(* IEC 61131-3 sources: SerComm/, 4 files *)

(* ---- SerComm.typ ---- *)
(********************************************************************
 * COPYRIGHT -- Automation Resources Group
 ********************************************************************
 * Library: SerComm
 * File: SerComm.typ
 * Author: David Blackburn
 * Created: June 21, 2013
 ********************************************************************
 * Data types of library SerComm
 ********************************************************************)

TYPE

END_TYPE

(* ---- SerialCommMgr.typ ---- *)
(*
 * File: SerialCommMgr.typ
 * Copyright (c) 2023 Loupe
 * https://loupe.team
 *
 * This file is part of SerComm, licensed under the MIT License.
 *
 *)

TYPE
	SERCOMM_ERR_enum :
		(
		SERCOMM_ERR_INVALIDINPUT := 50000,
		SERCOMM_ERR_RECVDATATOOLARGE,
		SERCOMM_ERR_SENDDATATOOLARGE,
		SERCOMM_ERR_
		);
	SERCOMM_ST_enum :
		(
		SERCOMM_ST_CLOSED,
		SERCOMM_ST_OPENING,
		SERCOMM_ST_RUNNING,
		SERCOMM_ST_CLOSING,
		SERCOMM_ST_ERROR
		);
	SERCOMM_RECV_ST_enum :
		(
		SERCOMM_RECV_ST_READ,
		SERCOMM_RECV_ST_RBUF
		);
	SERCOMM_SEND_ST_enum :
		(
		SERCOMM_SEND_ST_GBUF,
		SERCOMM_SEND_ST_IDLE,
		SERCOMM_SEND_ST_WRITE,
		SERCOMM_SEND_ST_ROBUF
		);
	SerialCommMgr_Int_FUB_typ : 	STRUCT
		Open : FRM_xopen;
		Read : FRM_read;
		ReleaseReadBuffer : FRM_rbuf;
		GetWriteBuffer : FRM_gbuf;
		Write : FRM_write;
		ReleaseWriteBuffer : FRM_robuf;
		Close : FRM_close;
	END_STRUCT;
	SerialCommMgr_Internal_typ : 	STRUCT
		CommState : SERCOMM_ST_enum;
		SendState : SERCOMM_SEND_ST_enum;
		ReceiveState : SERCOMM_RECV_ST_enum;
		FrameIdent : UDINT;
		WriteBuffer : UDINT;
		WriteBufferLength : UINT;
		CMD : SerialCommMgr_IN_CMD_typ;
		FUB : SerialCommMgr_Int_FUB_typ;
	END_STRUCT;
	SerialCommMgr_OUT_STAT_typ : 	STRUCT
		CommunicationActive : BOOL;
		DataSent : BOOL;
		NewDataAvailable : BOOL;
		Data : ARRAY[0..SERCOMM_MAI_DATA]OF USINT;
		DataLength : UDINT;
		Error : BOOL;
		ErrorID : UINT;
		ErrorString : STRING[SERCOMM_STRLEN_ERRORSTRING];
	END_STRUCT;
	SerialCommMgr_OUT_typ : 	STRUCT
		STAT : SerialCommMgr_OUT_STAT_typ;
	END_STRUCT;
	SerialCommMgr_IN_CFG_typ : 	STRUCT
		INADeviceName : STRING[SERCOMM_STRLEN_DEVICENAME] := 'IF1';
		Mode : STRING[SERCOMM_STRLEN_MODE];
		pConfig : UDINT;
	END_STRUCT;
	SerialCommMgr_IN_PAR_typ : 	STRUCT
		Data : ARRAY[0..SERCOMM_MAI_DATA]OF USINT;
		DataLength : UDINT;
		AllowContinuousSend : BOOL;
		AllowContinuousReceive : BOOL;
	END_STRUCT;
	SerialCommMgr_IN_CMD_typ : 	STRUCT
		Enable : BOOL;
		Send : BOOL;
		AcknowledgeData : BOOL;
		AcknowledgeError : BOOL;
	END_STRUCT;
	SerialCommMgr_IN_typ : 	STRUCT
		CMD : SerialCommMgr_IN_CMD_typ;
		PAR : SerialCommMgr_IN_PAR_typ;
		CFG : SerialCommMgr_IN_CFG_typ;
	END_STRUCT;
	SerialCommMgr_typ : 	STRUCT
		IN : SerialCommMgr_IN_typ;
		OUT : SerialCommMgr_OUT_typ;
		Internal : SerialCommMgr_Internal_typ;
	END_STRUCT;
END_TYPE

(* ---- SerComm.fun ---- *)
(*
 * File: SerComm.fun
 * Copyright (c) 2023 Loupe
 * https://loupe.team
 *
 * This file is part of SerComm, licensed under the MIT License.
 *
 *)

FUNCTION SerialCommFn_Cyclic : UINT (*Cyclic function for managing serial communications*)
	VAR_IN_OUT
		t : SerialCommMgr_typ;
	END_VAR
END_FUNCTION

FUNCTION SerialCommMgr : UINT (*Cyclic function for managing serial communications*)
	VAR_IN_OUT
		t : SerialCommMgr_typ;
	END_VAR
END_FUNCTION

FUNCTION SerialCommSend : UINT (*Cyclic function for managing serial communications*)
	VAR_IN_OUT
		t : SerialCommMgr_typ;
	END_VAR
END_FUNCTION

FUNCTION SerialCommReceive : UINT (*Cyclic function for managing serial communications*)
	VAR_IN_OUT
		t : SerialCommMgr_typ;
	END_VAR
END_FUNCTION

(* ---- SerComm.var ---- *)
(********************************************************************
 * COPYRIGHT -- Automation Resources Group
 ********************************************************************
 * Library: SerComm
 * File: SerComm.var
 * Author: David Blackburn
 * Created: June 21, 2013
 ********************************************************************
 * Constants of library SerComm
 ********************************************************************)
VAR CONSTANT
	SERCOMM_MAI_DATA : UINT := 255;
	SERCOMM_STRLEN_DEVICENAME : USINT := 80;
	SERCOMM_STRLEN_MODE : USINT := 255;
	SERCOMM_STRLEN_ERRORSTRING : USINT := 80;
END_VAR
